{attribute 'GeneratedUsingTerminal: EL9221-4030-0018'}
{attribute addProperty BoxType "EL9221-4030-0018"}
{attribute addProperty Id "ResetBOOL1SwitchBOOL1"}
{attribute addProperty CRC "1397746457"}
{attribute addProperty Size "2"}
TYPE Control_534FEB19 :
STRUCT
	{attribute addProperty Name "Reset"}
	Reset : BOOL;
	{attribute addProperty Name "Switch"}
	Switch : BOOL;
END_STRUCT
END_TYPE

(* stored: Version 1.2.0.0, ProductVersion 3.1.4024.9
   DUT Control_534FEB19: Id {88a7eb13-aa1a-49af-941d-fc8fa1c88554} *)
